// TIA Portal V20 export
// export: Created 2026-10-06T14:30:21.2976712Z, ExportSetting WithDefaults, DisplayName Totally Integrated Automation Portal, DisplayVersion V20, DisplayName TIA Portal Openness, DisplayVersion V20, DisplayName TIA Portal Version Control Interface, DisplayVersion V20, DisplayName SINAMICS Startdrive Advanced, DisplayVersion V20, DisplayName SINAMICS Startdrive G130, G150, S120, S150, SINAMICS MV, G220, S200, S210, DisplayVersion V20, DisplayName SINAMICS Startdrive G110M, G120, G120C, G120D, G120P, G115D, DisplayVersion V20, DisplayName STEP 7 Professional, DisplayVersion V20, DisplayName STEP 7 Safety, DisplayVersion V20, DisplayName WinCC Basic/Comfort/Advanced, DisplayVersion V20, DisplayName WinCC Unified, DisplayVersion V20
FUNCTION_BLOCK "MotorGroups"   // FB3, LAD
{ S7_Optimized_Access := 'TRUE' }
VERSION : 0.1
// stored: AutoNumber false, IsIECCheckEnabled false, IsRetainMemResEnabled false, MemoryReserve 100, SetENOAutomatically false, UDAEnableTagReadback false
   VAR
      Group1 { S7_SetPoint := 'True'} : "MotorSequenceLAD";
      Group2 { S7_SetPoint := 'True'} : "MotorSequenceLAD";
   END_VAR
BEGIN

REGION Network 1
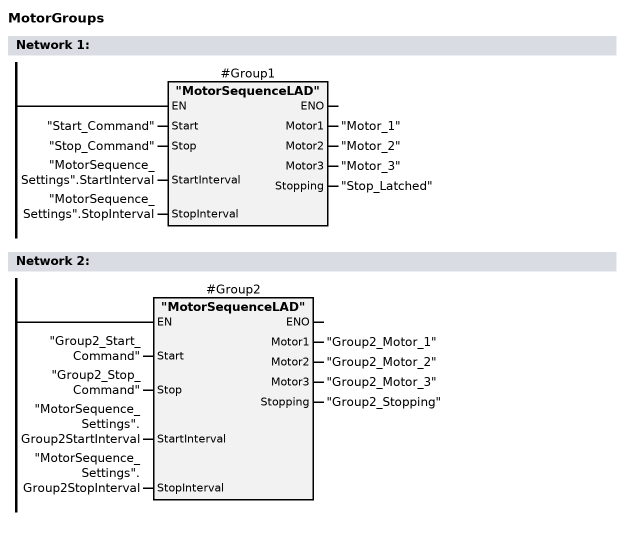
   RUNG wire#powerrail
      #Group1(Start := "Start_Command", Stop := "Stop_Command", StartInterval := "MotorSequence_Settings".StartInterval, StopInterval := "MotorSequence_Settings".StopInterval, Motor1 => "Motor_1", Motor2 => "Motor_2", Motor3 => "Motor_3", Stopping => "Stop_Latched")
   END_RUNG
   // the same network as SCL:
   #Group1(Start := "Start_Command",   // "MotorSequenceLAD"
           Stop := "Stop_Command",
           StartInterval := "MotorSequence_Settings".StartInterval,
           StopInterval := "MotorSequence_Settings".StopInterval,
           Motor1 => "Motor_1",
           Motor2 => "Motor_2",
           Motor3 => "Motor_3",
           Stopping => "Stop_Latched");
END_REGION

REGION Network 2
   RUNG wire#powerrail
      #Group2(Start := "Group2_Start_Command", Stop := "Group2_Stop_Command", StartInterval := "MotorSequence_Settings".Group2StartInterval, StopInterval := "MotorSequence_Settings".Group2StopInterval, Motor1 => "Group2_Motor_1", Motor2 => "Group2_Motor_2", Motor3 => "Group2_Motor_3", Stopping => "Group2_Stopping")
   END_RUNG
   // the same network as SCL:
   #Group2(Start := "Group2_Start_Command",   // "MotorSequenceLAD"
           Stop := "Group2_Stop_Command",
           StartInterval := "MotorSequence_Settings".Group2StartInterval,
           StopInterval := "MotorSequence_Settings".Group2StopInterval,
           Motor1 => "Group2_Motor_1",
           Motor2 => "Group2_Motor_2",
           Motor3 => "Group2_Motor_3",
           Stopping => "Group2_Stopping");
END_REGION
END_FUNCTION_BLOCK
